(* CoDeSys 2.3.9.41 project: rePlc160.pro *)
(* Libraries: STANDARD.LIB 4.10.05 10:14:46, SmsOwenLib.lib 5.10.12 16:48:36, IECSFC.LIB 13.4.06 14:51:28, Util.lib 18.5.10 15:14:28, SysLibCom.lib 20.2.06 13:31:08, UNM.lib 14.2.06 12:27:08, SMS.lib 29.7.11 08:51:48, SYSLIBTIME.LIB 20.2.06 13:31:16, SYSTASKINFO.LIB 20.2.06 13:31:38, ANALYZATION.LIB 5.10.99 08:05:06, SYSLIBCALLBACK.LIB 20.2.06 13:31:08 *)

(* PLC configuration (modules and I/O channels)
DI_leakSens1 AT %IX0.0 [BitInput] Discrete input 1
DI_leakSens2 AT %IX0.1 [BitInput] Discrete input 2
DI_lamp1 AT %IX0.2 [BitInput] Discrete input 3
DI_lamp2 AT %IX0.3 [BitInput] Discrete input 4
AT %IB1.0 [ByteInput] DI_POLIW
AT %IB1.1 [ByteInput] DI_FOUNTAIN
AT %QB2.0 [ByteOutput] DO_POLIW_FOUN_LEAK
AT %QB2.1 [ByteOutput] DO_FOUN
AI_pres AT %IR3.0 [FloatInputP] AI #1 {AIN_TYPE = 0-20 mA; Peak_Filtr = 200; Flt_Ch = Off; TauRC = 10; MinFV = 0; MaxFV = 20000.0}
AI_level AT %IR3.1 [FloatInputP] AI #2 {AIN_TYPE = 0-20 mA; Peak_Filtr = 200; Flt_Ch = Off; TauRC = 10; MinFV = 0; MaxFV = 20000.0}
AI_T1 AT %IR3.2 [FloatInputP] AI #3 {AIN_TYPE = 4-20 mA; Peak_Filtr = 200; Flt_Ch = Off; TauRC = 10; MinFV = 0; MaxFV = 20000.0}
AI_T2 AT %IR3.3 [FloatInputP] AI #4 {AIN_TYPE = 4-20 mA; Peak_Filtr = 200; Flt_Ch = Off; TauRC = 10; MinFV = 0; MaxFV = 20000.0}
AI_05 AT %IR3.4 [FloatInputP] AI #5 {AIN_TYPE = 0-20 mA; Peak_Filtr = 200; Flt_Ch = Off; TauRC = 10; MinFV = 0; MaxFV = 20000.0}
AI_06 AT %IR3.5 [FloatInputP] AI #6 {AIN_TYPE = 0-20 mA; Peak_Filtr = 200; Flt_Ch = Off; TauRC = 10; MinFV = 0; MaxFV = 20000.0}
AI_volt AT %IR3.6 [FloatInputP] AI #7 {AIN_TYPE = 0-20 mA; Peak_Filtr = 200; Flt_Ch = Off; TauRC = 10; MinFV = 0; MaxFV = 20000.0}
AI_08 AT %IR3.7 [FloatInputP] AI #8 {AIN_TYPE = 0-20 mA; Peak_Filtr = 200; Flt_Ch = Off; TauRC = 10; MinFV = 0; MaxFV = 20000.0}
AT %IW3.8 [WordInput] AI read time (10ms)
AO_fc AT %QR4.0 [FloatOutputP] AO #1 {AOUT_TYPE = 0-10V; SafeValueREAL = 0.0}
AO_dim1 AT %QR4.1 [FloatOutputP] AO #2 {AOUT_TYPE = 0-10V; SafeValueREAL = 0.0}
AO_dim2 AT %QR4.2 [FloatOutputP] AO #3 {AOUT_TYPE = 0-10V; SafeValueREAL = 0.0}
AO_dim3 AT %QR4.3 [FloatOutputP] AO #4 {AOUT_TYPE = 0-10V; SafeValueREAL = 0.0}
Special input [ID103] node 5, in %IB5 out %QB5 {Filtrationtime = 1000; PinCount = 1; WatchDogPeriod = 400; PollPeriod = 3000; Visibility = No}
  AT %IX5.0 [BitInput] Special input
Special output [ID104] node 6, in %IB6 out %QB6 {Visibility = No; PinCount = 1}
  AT %QX6.0 [BitOutput] Special output
Universal network module [UNM_ID300] node 7, in %IB7 out %QB7 {Visibility = No}
  RS-232 [COM2_USART] node 0, in %IB7.0 out %QB7.0 {CommunicationSpeed = 9600; Parity = NO PARITY CHECK; BitLength = 8 bits; StopLength = One stop bit; InterfaceType = RS232; FrameOriented = ASCII; Timeout = 0; Visibility = No}
AT %QB8.0.0.0 [ByteOutput] Line Status
AT %QB8.0.0.1 [ByteOutput] Modem Fault
startGPRS AT %QB8.0.0.2 [ByteOutput] Start_Auto_Dial
stopGPRG AT %QB8.0.0.3 [ByteOutput] Stop_Dial
RS-232 [COM2_USART] node 0, in %IB8.0.0.0 out %QB8.0.0.0 {CommunicationSpeed = 9600; Parity = NO PARITY CHECK; BitLength = 8 bits; StopLength = One stop bit; InterfaceType = RS232; FrameOriented = ASCII; Timeout = 0; Visibility = No}
PPP_Driver [PPP] node 1, in %IB8.0.0.1 out %QB8.0.0.1 {LoginString = mts; PasswordString = mts}
TCP [TCP_ID221] node 1, in %IB8.0.1 out %QB8.0.1 {RemotePort = 502; Visibility = No}
pad_PoliwDIST AT %QW8.1.0 [WordOutput]
pad_PoliwTELE AT %QW8.2.0 [WordOutput]
cir1On AT %QW8.3.0 [WordOutput]
cir1Off AT %QW8.4.0 [WordOutput]
cir2On AT %QW8.5.0 [WordOutput]
2 byte [Register] node 6, in %IB8.6 out %QB8.6
  cir2Off AT %QW8.6.0 [WordOutput]
2 byte [Register] node 7, in %IB8.7 out %QB8.7
  cir3On AT %QW8.7.0 [WordOutput]
2 byte [Register] node 8, in %IB8.8 out %QB8.8
  cir3Off AT %QW8.8.0 [WordOutput]
  FounDIST AT %QW8.9.0 [WordOutput]
  dist_staticFValue AT %QW8.10.0 [WordOutput]
  FounTELE AT %QW8.11.0 [WordOutput]
  p1 AT %QW8.12.0 [WordOutput]
  p2 AT %QW8.13.0 [WordOutput]
2 byte [Register] node 14, in %IB8.14 out %QB8.14
  p3 AT %QW8.14.0 [WordOutput]
2 byte [Register] node 15, in %IB8.15 out %QB8.15
  p4 AT %QW8.15.0 [WordOutput]
2 byte [Register] node 16, in %IB8.16 out %QB8.16
  p5 AT %QW8.16.0 [WordOutput]
2 byte [Register] node 17, in %IB8.17 out %QB8.17
  p6 AT %QW8.17.0 [WordOutput]
2 byte [Register] node 18, in %IB8.18 out %QB8.18
  p7 AT %QW8.18.0 [WordOutput]
2 byte [Register] node 19, in %IB8.19 out %QB8.19
  p8 AT %QW8.19.0 [WordOutput]
2 byte [Register] node 20, in %IB8.20 out %QB8.20
  p9 AT %QW8.20.0 [WordOutput]
  p10 AT %QW8.21.0 [WordOutput]
2 byte [Register] node 22, in %IB8.22 out %QB8.22
  T_STATE AT %QW8.22.0 [WordOutput]
2 byte [Register] node 23, in %IB8.23 out %QB8.23
  pad_t1 AT %QW8.23.0 [WordOutput]
2 byte [Register] node 24, in %IB8.24 out %QB8.24
  pad_t2 AT %QW8.24.0 [WordOutput]
2 byte [Register] node 25, in %IB8.25 out %QB8.25
  pad_t1_currSetTop AT %QW8.25.0 [WordOutput]
2 byte [Register] node 26, in %IB8.26 out %QB8.26
  pad_t1_currSetBottom AT %QW8.26.0 [WordOutput]
2 byte [Register] node 27, in %IB8.27 out %QB8.27
  pad_t2_currSetTop AT %QW8.27.0 [WordOutput]
2 byte [Register] node 28, in %IB8.28 out %QB8.28
  pad_t2_currSetBottom AT %QW8.28.0 [WordOutput]
2 byte [Register] node 29, in %IB8.29 out %QB8.29
  pad_t1_day AT %QW8.29.0 [WordOutput]
2 byte [Register] node 30, in %IB8.30 out %QB8.30
  pad_t1_night AT %QW8.30.0 [WordOutput]
2 byte [Register] node 31, in %IB8.31 out %QB8.31
  pad_t2_day AT %QW8.31.0 [WordOutput]
2 byte [Register] node 32, in %IB8.32 out %QB8.32
  pad_t2_night AT %QW8.32.0 [WordOutput]
2 byte [Register] node 33, in %IB8.33 out %QB8.33
  pad_t1_daySetTop AT %QW8.33.0 [WordOutput]
2 byte [Register] node 34, in %IB8.34 out %QB8.34
  pad_t1_daySetBottom AT %QW8.34.0 [WordOutput]
2 byte [Register] node 35, in %IB8.35 out %QB8.35
  pad_t1_nightSetTop AT %QW8.35.0 [WordOutput]
2 byte [Register] node 36, in %IB8.36 out %QB8.36
  pad_t1_nightSetBottom AT %QW8.36.0 [WordOutput]
2 byte [Register] node 37, in %IB8.37 out %QB8.37
  pad_t2_daySetTop AT %QW8.37.0 [WordOutput]
2 byte [Register] node 38, in %IB8.38 out %QB8.38
  pad_t2_daySetBottom AT %QW8.38.0 [WordOutput]
  pad_t2_nightSetTop AT %QW8.39.0 [WordOutput]
  pad_t2_nightSetBottom AT %QW8.40.0 [WordOutput]
  pad_sens1_4ma AT %QW8.41.0 [WordOutput]
  pad_sens1_20ma AT %QW8.42.0 [WordOutput]
  pad_sens2_4ma AT %QW8.43.0 [WordOutput]
  pad_sens2_20ma AT %QW8.44.0 [WordOutput]
  dim1 AT %QW8.45.0 [WordOutput]
  dim2 AT %QW8.46.0 [WordOutput]
  dim3 AT %QW8.47.0 [WordOutput]
  RESERVE_1 AT %QW8.48.0 [WordOutput]
  RESERVE_2 AT %QW8.49.0 [WordOutput]
  weBITS_IN AT %QW8.50.0 [WordOutput] (leak)
  weBITS_OUT AT %QW8.51.0 [WordOutput] leakSens1,leakSens2,valveStat,drePumpStat,unknPump
  dist_LAMP AT %QW8.52.0 [WordOutput]
  tele_LAMP AT %QW8.53.0 [WordOutput]
  lamp1On AT %QW8.54.0 [WordOutput]
  lamp1Off AT %QW8.55.0 [WordOutput]
  lamp2On AT %QW8.56.0 [WordOutput]
  lamp2Off AT %QW8.57.0 [WordOutput]
  lamp3On AT %QW8.58.0 [WordOutput]
  lamp3Off AT %QW8.59.0 [WordOutput]
  year AT %QW8.60.0 [WordOutput]
  monthday AT %QW8.61.0 [WordOutput]
  hourminute AT %QW8.62.0 [WordOutput]
  tele_year AT %QW8.63.0 [WordOutput]
  tele_month AT %QW8.64.0 [WordOutput]
  tele_day AT %QW8.65.0 [WordOutput]
  tele_hour AT %QW8.66.0 [WordOutput]
  tele_minute AT %QW8.67.0 [WordOutput]
  dist_dom2 AT %QW8.68.0 [WordOutput]
  tele_dom2 AT %QW8.69.0 [WordOutput]
  tele_pres AT %QW8.70.0 [WordOutput]
  tele_level AT %QW8.71.0 [WordOutput]
  tele_voltage AT %QW8.72.0 [WordOutput]
*)

(* Global variable list: Global_Variables *)
VAR_GLOBAL

(* Times *)
	GetTime: CurTimeEx;
	TimeAndDate: SystemTimeDate;
	Sys_Time: SysTime64;

	SMS_ID  : WORD;

	DI_door : BOOL := FALSE;
	DO_door : BOOL := FALSE;
	DO_drePump : BOOL := FALSE;
	DO_unknownPump : BOOL := FALSE;
	DI_staticMode : BOOL := FALSE;
	DI_dynamicMode : BOOL := FALSE;
	DI_v1_manMode : BOOL := FALSE;
	DI_v2_manMode : BOOL := FALSE;
	DI_v3_manMode : BOOL := FALSE;
	DO_pump : BOOL := FALSE;
	DI_pumpState : BOOL := FALSE;

END_VAR

(* POU PLC_PRG, ST *)
PROGRAM PLC_PRG
VAR
	NO_FIRST_PASS : BOOL;
END_VAR
VAR RETAIN
	weBITS_IN_save : WORD;
END_VAR
IF NO_FIRST_PASS = FALSE
	THEN _WithdrawRetain;
	NO_FIRST_PASS := TRUE;
END_IF;

_CheckNewValue;

_Leakage;

_Tele;

POLIW;

FOUNTAIN;

TEMPERATURE;

LIGHT;

SMS;

DOM2;
END_PROGRAM
ACTION _CheckNewValue:
IF weBITS_IN_save <> weBITS_IN
	THEN weBITS_IN_save := weBITS_IN;
END_IF;
END_ACTION
ACTION _Leakage:
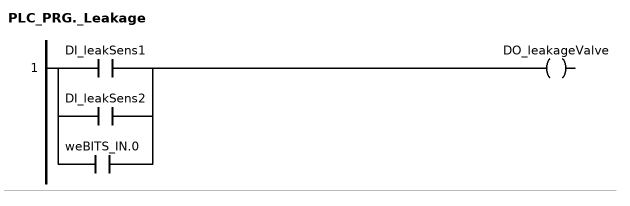
_LD_ (* Ladder Diagram *)
NETWORK 1
	{ [DI_leakSens1] | [DI_leakSens2] | [weBITS_IN.0] } --- (DO_leakageValve)
_END_LD_
(* the same logic as Structured Text *)
(* Network 1 *)
DO_leakageValve := DI_leakSens1 OR DI_leakSens2 OR weBITS_IN.0;
END_ACTION
ACTION _Tele:
weBITS_OUT.0 := DI_leakSens1;
weBITS_OUT.1 := DI_leakSens2;
weBITS_OUT.2 := DO_leakageValve;

(*
AI1_OUT := REAL_TO_WORD ( AI_01 );
AI2_OUT := REAL_TO_WORD ( AI_02 );
AI3_OUT := REAL_TO_WORD ( AI_T1 );
AI4_OUT := REAL_TO_WORD ( AI_T2 );
AI5_OUT := REAL_TO_WORD ( AI_05 );
AI6_OUT := REAL_TO_WORD ( AI_06 );
AI7_OUT := REAL_TO_WORD ( AI_07 );
AI8_OUT := REAL_TO_WORD ( AI_08 );
*)
(*
someDIs.0 := DI_konduk;
someDIs.1 := DI_powerSupply;
someDIs.2 := DI_banya;
someDIs.3 := DI_pool;
someDIs.4 := DI_foun;
someDIs.5 := DI_poliw;
someDIs.6 := DO_door;
*)
END_ACTION
ACTION _WithdrawRetain:
weBITS_IN := weBITS_IN_save;
END_ACTION

(* POU POLIW, ST *)
PROGRAM POLIW
VAR
	NO_FIRST_PASS : BOOL;
	PUNCH : WORD;
	setYear : INT;
	setMonth, setDay, setHour, setMinute : BYTE;
	set_time : BOOL;

(* bits *)
	dist_valve1, dist_valve2, dist_valve3 : BOOL;

	dist_manka : BOOL;

	MON : BOOL;
	TUE : BOOL;
	WED : BOOL;
	THU : BOOL;
	FRI : BOOL;
	SAT : BOOL;
	SUN : BOOL;

	cir1OnHH, cir1OnMM, cir1OffHH, cir1OffMM,
	cir2OnHH, cir2OnMM, cir2OffHH, cir2OffMM,
	cir3OnHH, cir3OnMM, cir3OffHH, cir3OffMM : BYTE;


	tele_pumpState, tele_v1state, tele_v2state, tele_v3state,
	tele_rainSens, tele_humSens : BOOL;

	cir1mustRun: BOOL;
	cir2mustRun: BOOL;
	cir3mustRun: BOOL;
	dayOk: BOOL;

	waterFault: BOOL;

	auto_pump_start: BOOL;
	auto_v1_open: BOOL;
	auto_v2_open: BOOL;
	auto_v3_open: BOOL;

	dist_pump_start: BOOL;
	dist_v1_open: BOOL;
	dist_v2_open: BOOL;
	dist_v3_open: BOOL;

	v1_auto_started: BOOL;
	FN_dist_v1_off: F_TRIG;
	v1_must_dist_stop: BOOL;
	v2_auto_started: BOOL;
	FN_dist_v2_off: F_TRIG;
	v2_must_dist_stop: BOOL;
	v3_auto_started: BOOL;
	FN_dist_v3_off: F_TRIG;
	v3_must_dist_stop: BOOL;
END_VAR

VAR RETAIN
	SAVE_BITS : WORD;

	save_cir1On, save_cir1Off,
       save_cir2On, save_cir2Off,
	 save_cir3On, save_cir3Off  : WORD;

	save_year, save_monthday, save_hourminute : WORD;
END_VAR
(* 				first pass 				*)
IF NO_FIRST_PASS = FALSE
	THEN WithdrawRetain;
	PUNCH := 65535;
	Obtaining;
	PUNCH := 0;
	NO_FIRST_PASS := TRUE;
END_IF;

(*			    main cycle		  		*)
PUNCH := 0;

set_time := weBITS_IN.1;
Times; (* получение текущего времени *)

CheckNewVal; (* проверка наличия новых значений переменных из модбас *)
				 (* и запись их в retain переменные *)
IF PUNCH > 0 THEN
	Obtaining; (* распаковка retain переменных в рабочие переменные *)
END_IF;

Schedule; (* основной цикл полива *)
(*
ExMech; (* управление исполнительным механизмом *)
*)
Outs; (* управление выходами контроллера на полив *)

HandOff;
Tele; (* передача рабочего состояния на верхний уровень *)
END_PROGRAM
ACTION CheckNewVal:
IF SAVE_BITS <> pad_PoliwDIST
	THEN SAVE_BITS := pad_PoliwDIST;
			PUNCH.0 := TRUE;
END_IF;



IF save_cir1On <> cir1On
	THEN save_cir1On := cir1On;
			PUNCH.1 := TRUE;
END_IF;

IF save_cir1Off <> cir1Off
	THEN save_cir1Off := cir1Off;
			PUNCH.2 := TRUE;
END_IF;


IF save_cir2On <> cir2On
	THEN save_cir2On := cir2On;
			PUNCH.3 := TRUE;
END_IF;

IF save_cir2Off <> cir2Off
	THEN save_cir2Off := cir2Off;
			PUNCH.4 := TRUE;
END_IF;


IF save_cir3On <> cir3On
	THEN save_cir3On := cir3On;
			PUNCH.5 := TRUE;
END_IF;

IF save_cir3Off <> cir3Off
	THEN save_cir3Off := cir3Off;
			PUNCH.6 := TRUE;
END_IF;


IF save_year <> year
	THEN save_year := year;
			PUNCH.9 := TRUE;
END_IF;

IF save_monthday <> monthday
	THEN save_monthday := monthday;
			PUNCH.10 := TRUE;
END_IF;

IF save_hourminute <> hourminute
	THEN save_hourminute := hourminute;
			PUNCH.11 := TRUE;
END_IF;
END_ACTION
ACTION HandOff:
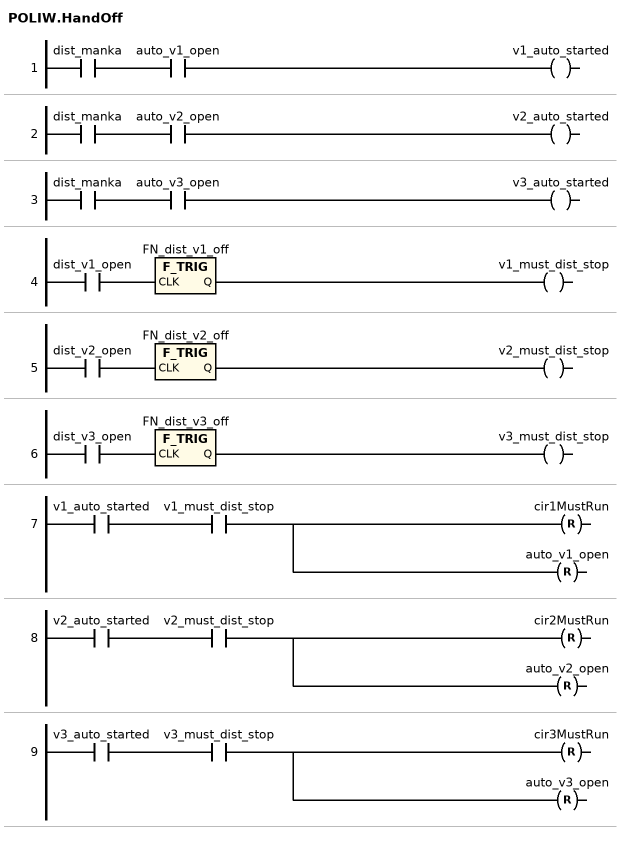
_LD_ (* Ladder Diagram *)
NETWORK 1
	[dist_manka] - [auto_v1_open] --- (v1_auto_started)
NETWORK 2
	[dist_manka] - [auto_v2_open] --- (v2_auto_started)
NETWORK 3
	[dist_manka] - [auto_v3_open] --- (v3_auto_started)
NETWORK 4
	[dist_v1_open] - FN_dist_v1_off:F_TRIG(CLK: *) --- (v1_must_dist_stop)
NETWORK 5
	[dist_v2_open] - FN_dist_v2_off:F_TRIG(CLK: *) --- (v2_must_dist_stop)
NETWORK 6
	[dist_v3_open] - FN_dist_v3_off:F_TRIG(CLK: *) --- (v3_must_dist_stop)
NETWORK 7
	[v1_auto_started] - [v1_must_dist_stop] --- (R cir1MustRun) (R auto_v1_open)
NETWORK 8
	[v2_auto_started] - [v2_must_dist_stop] --- (R cir2MustRun) (R auto_v2_open)
NETWORK 9
	[v3_auto_started] - [v3_must_dist_stop] --- (R cir3MustRun) (R auto_v3_open)
_END_LD_
(* the same logic as Structured Text *)
(* Network 1 *)
v1_auto_started := dist_manka AND auto_v1_open;
(* Network 2 *)
v2_auto_started := dist_manka AND auto_v2_open;
(* Network 3 *)
v3_auto_started := dist_manka AND auto_v3_open;
(* Network 4 *)
FN_dist_v1_off(CLK := dist_v1_open);
v1_must_dist_stop := FN_dist_v1_off.Q;
(* Network 5 *)
FN_dist_v2_off(CLK := dist_v2_open);
v2_must_dist_stop := FN_dist_v2_off.Q;
(* Network 6 *)
FN_dist_v3_off(CLK := dist_v3_open);
v3_must_dist_stop := FN_dist_v3_off.Q;
(* Network 7 *)
IF v1_auto_started AND v1_must_dist_stop THEN cir1MustRun := FALSE; auto_v1_open := FALSE; END_IF;
(* Network 8 *)
IF v2_auto_started AND v2_must_dist_stop THEN cir2MustRun := FALSE; auto_v2_open := FALSE; END_IF;
(* Network 9 *)
IF v3_auto_started AND v3_must_dist_stop THEN cir3MustRun := FALSE; auto_v3_open := FALSE; END_IF;
END_ACTION
ACTION Obtaining:
IF PUNCH.0 THEN
	dist_manka := SAVE_BITS.0;
	dist_valve1 := SAVE_BITS.1;
	dist_valve2 := SAVE_BITS.2;
	dist_valve3 := SAVE_BITS.3;

	MON := SAVE_BITS.6;
	TUE := SAVE_BITS.7;
	WED := SAVE_BITS.8;
	THU := SAVE_BITS.9;
	FRI := SAVE_BITS.10;
	SAT := SAVE_BITS.11;
	SUN := SAVE_BITS.12;

	PUNCH.0 := FALSE;
END_IF;

(*
	lo,hi : byte
	w : word

	lo := word_to_byte(w)
	hi := word_to_byte(w/256)
	w := 256*hi + lo 
*)

IF PUNCH.1 THEN
	cir1OnHH := WORD_TO_BYTE ( save_cir1On );
	cir1OnMM := WORD_TO_BYTE ( save_cir1On / 256 );
	PUNCH.1 := FALSE;
END_IF;

IF PUNCH.2 THEN
	cir1OffHH := WORD_TO_BYTE ( save_cir1Off );
	cir1OffMM := WORD_TO_BYTE ( save_cir1Off / 256 );
	PUNCH.2 := FALSE;
END_IF;

IF PUNCH.3 THEN
	cir2OnHH := WORD_TO_BYTE ( save_cir2On );
	cir2OnMM := WORD_TO_BYTE ( save_cir2On / 256 );
	PUNCH.3 := FALSE;
END_IF;

IF PUNCH.4 THEN
	cir2OffHH := WORD_TO_BYTE ( save_cir2Off );
	cir2OffMM := WORD_TO_BYTE ( save_cir2Off / 256 );
	PUNCH.4 := FALSE;
END_IF;

IF PUNCH.5 THEN
	cir3OnHH := WORD_TO_BYTE ( save_cir3On );
	cir3OnMM := WORD_TO_BYTE ( save_cir3On / 256 );
	PUNCH.5 := FALSE;
END_IF;

IF PUNCH.6 THEN
	cir3OffHH := WORD_TO_BYTE ( save_cir3Off );
	cir3OffMM := WORD_TO_BYTE ( save_cir3Off / 256 );
	PUNCH.6 := FALSE;
END_IF;


IF PUNCH.9 THEN
	setYear := WORD_TO_INT ( save_year );
	PUNCH.9 := FALSE;
END_IF;


IF PUNCH.10 THEN
	setDay := WORD_TO_BYTE ( save_monthday );
	setMonth := WORD_TO_BYTE ( save_monthday / 256 );
	PUNCH.10 := FALSE;
END_IF;

IF PUNCH.11 THEN
	setMinute := WORD_TO_BYTE ( save_hourminute );
	setHour := WORD_TO_BYTE ( save_hourminute / 256 );
	PUNCH.11 := FALSE;
END_IF;
END_ACTION
ACTION Outs:
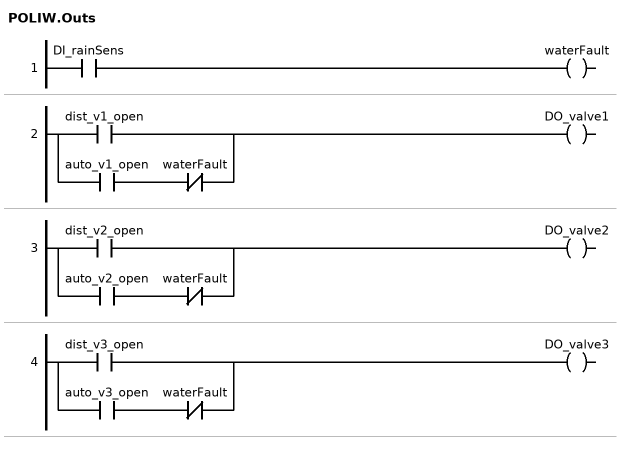
_LD_ (* Ladder Diagram *)
NETWORK 1
	[DI_rainSens] --- (waterFault)
NETWORK 2
	{ [dist_v1_open] | [auto_v1_open] - [/waterFault] } --- (DO_valve1)
NETWORK 3
	{ [dist_v2_open] | [auto_v2_open] - [/waterFault] } --- (DO_valve2)
NETWORK 4
	{ [dist_v3_open] | [auto_v3_open] - [/waterFault] } --- (DO_valve3)
_END_LD_
(* the same logic as Structured Text *)
(* Network 1 *)
waterFault := DI_rainSens;
(* Network 2 *)
DO_valve1 := dist_v1_open OR auto_v1_open AND NOT waterFault;
(* Network 3 *)
DO_valve2 := dist_v2_open OR auto_v2_open AND NOT waterFault;
(* Network 4 *)
DO_valve3 := dist_v3_open OR auto_v3_open AND NOT waterFault;
END_ACTION
ACTION Schedule:
(* контур 1 *)
IF ( cir1OnHH = TimeAndDate.Hour ) AND ( cir1OnMM = TimeAndDate.Minute ) AND ( TimeAndDate.Second = 0 )
	THEN cir1mustRun := TRUE;
END_IF;

IF ( cir1OffHH = TimeAndDate.Hour ) AND ( cir1OffMM = TimeAndDate.Minute ) AND ( TimeAndDate.Second = 0 )
	THEN cir1mustRun := FALSE;
END_IF;

(* контур 2 *)
IF ( cir2OnHH = TimeAndDate.Hour ) AND ( cir2OnMM = TimeAndDate.Minute ) AND ( TimeAndDate.Second = 0 )
	THEN cir2mustRun := TRUE;
END_IF;

IF ( cir2OffHH = TimeAndDate.Hour ) AND ( cir2OffMM = TimeAndDate.Minute ) AND ( TimeAndDate.Second = 0 )
	THEN cir2mustRun := FALSE;
END_IF;

(* контур 3 *)
IF ( cir3OnHH = TimeAndDate.Hour ) AND ( cir3OnMM = TimeAndDate.Minute ) AND ( TimeAndDate.Second = 0 )
	THEN cir3mustRun := TRUE;
END_IF;

IF ( cir3OffHH = TimeAndDate.Hour ) AND ( cir3OffMM = TimeAndDate.Minute ) AND ( TimeAndDate.Second = 0 )
	THEN cir3mustRun := FALSE;
END_IF;

(* день недели *)
CASE TimeAndDate.DayOfWeek OF
	1 : IF MON
	     	THEN dayOk := TRUE;
		ELSE dayOk := FALSE;
	     END_IF;

	2 : IF TUE
	     	THEN dayOk := TRUE;
		ELSE dayOk := FALSE;
	     END_IF;

      3 : IF WED
	     	THEN dayOk := TRUE;
		ELSE dayOk := FALSE;
	     END_IF;

      4 : IF THU
	     	THEN dayOk := TRUE;
		ELSE dayOk := FALSE;
	     END_IF;

      5 : IF FRI
	     	THEN dayOk := TRUE;
		ELSE dayOk := FALSE;
	     END_IF;

      6 : IF SAT
	     	THEN dayOk := TRUE;
		ELSE dayOk := FALSE;
	     END_IF;

      0 : IF SUN
	     	THEN dayOk := TRUE;
		ELSE dayOk := FALSE;
	     END_IF;
END_CASE;

(* авто *)
IF dist_manka = FALSE THEN
	(* клапана *)
	IF ( cir1mustRun ) AND ( dayOk )
		THEN auto_v1_open := TRUE;
		ELSE auto_v1_open := FALSE;
	END_IF;

	IF ( cir2mustRun ) AND ( dayOk )
		THEN auto_v2_open := TRUE;
		ELSE auto_v2_open := FALSE;
	END_IF;

	IF ( cir3mustRun ) AND ( dayOk )
		THEN auto_v3_open := TRUE;
		ELSE auto_v3_open := FALSE;
	END_IF;
END_IF;

(* ручное дистанционно *)
IF dist_manka  THEN
	IF dist_valve1
		THEN dist_v1_open := TRUE;
		ELSE dist_v1_open := FALSE;
	END_IF;

	IF dist_valve2
		THEN dist_v2_open := TRUE;
		ELSE dist_v2_open := FALSE;
	END_IF;

	IF dist_valve3
		THEN dist_v3_open := TRUE;
		ELSE dist_v3_open := FALSE;
	END_IF;
END_IF;

(* примечание: помимо дистанционного управления есть управление с галетников,
				   имеющее наивысший приоритет.
 				   управление с галетников описано в Outs 						

уже нет		*)
END_ACTION
ACTION Tele:
(*pad_PoliwTELE.0 := DI_pumpState;*)
pad_PoliwTELE.1 := DO_valve1;
pad_PoliwTELE.2 := DO_valve2;
pad_PoliwTELE.3 := DO_valve3;
(*pad_PoliwTELE.4 := DO_valve4;
pad_PoliwTELE.5 := DO_exMech;*)
pad_PoliwTELE.6 := DI_rainSens;
(*pad_PoliwTELE.7 := DI_humSens;*)

tele_year := TimeAndDate.Year;
tele_month := TimeAndDate.Month;
tele_day := TimeAndDate.Day;
tele_hour := TimeAndDate.Hour;
tele_minute := TimeAndDate.Minute;
END_ACTION
ACTION Times:
TimeAndDate.Day :=0;
TimeAndDate.DayOfWeek :=0;
TimeAndDate.dwHighMsec :=0;
TimeAndDate.dwLowMSecs :=0;
TimeAndDate.Milliseconds :=0;
TimeAndDate.Minute :=0;
TimeAndDate.Second :=0;
TimeAndDate.Hour :=0;
TimeAndDate.Year :=0;
TimeAndDate.Month :=0;
Sys_time.ulHigh :=0;
Sys_time.ulLow :=0;
GetTime (SystemTime:=Sys_Time , TimeDate:= TimeAndDate);


IF set_time THEN

	TimeAndDate.Minute:=setMinute;
	TimeAndDate.Second:=0;
	TimeAndDate.Hour:=setHour;
	TimeAndDate.Day:=setDay;
	TimeAndDate.Month:=setMonth;
	TimeAndDate.Year:=setYear;
	GetTime (SystemTime:=Sys_Time , TimeDate:= TimeAndDate);

END_IF;
END_ACTION
ACTION WithdrawRetain:
pad_PoliwDIST := SAVE_BITS;

cir1On := save_cir1On;
cir1Off := save_cir1Off;

cir2On := save_cir2On;
cir2Off := save_cir2Off;

cir3On := save_cir3On;
cir3Off := save_cir3Off;
END_ACTION

(* POU FOUNTAIN, ST *)
PROGRAM FOUNTAIN
VAR
	NO_FIRST_PASS : BOOL;
	PUNCH : WORD;

	tele_byte : BYTE;

	dist_founOn, dist_dynamic : BOOL;

	M1: BOOL;
	founT1: TON;
	M2: BOOL;
	founT2: TON;
	M3: BOOL;
	founT3: TON;
	M4: BOOL;
	founT4: TON;
	M5: BOOL;
	founT5: TON;
	M6: BOOL;
	founT6: TON;
	M7: BOOL;
	founT7: TON;
	M8: BOOL;
	founT8: TON;
	M9: BOOL;
	founT9: TON;
	M10: BOOL;
	founT10: TON;

	nodyn: BOOL;

	FPFON: R_TRIG;

	galetMode: BOOL;

(* ex-ratain*)
	staticFValue : REAL;

	founV1F: REAL;
	founV2F: REAL;
	founV3F: REAL;
	founV4F: REAL;
	founV5F: REAL;
	founV6F: REAL;
	founV7F: REAL;
	founV8F: REAL;
	founV9F: REAL;
	founV10F: REAL;

	founS1T: TIME;
	founS2T: TIME;
	founS3T: TIME;
	founS4T: TIME;
	founS5T: TIME;
	founS6T: TIME;
	founS7T: TIME;
	founS8T: TIME;
	founS9T: TIME;
	founS10T: TIME;
END_VAR

VAR RETAIN
	save_DIST : WORD;
	save_staticFValue : WORD;
	save_p1, save_p2, save_p3, save_p4, save_p5,
	save_p6, save_p7, save_p8, save_p9, save_p10 : WORD;

END_VAR
VAR (* helpers for the ST form of the networks *)
	_p1 : BOOL;
	_p2 : BOOL;
	_p3 : BOOL;
	_p4 : BOOL;
	_p5 : BOOL;
	_p6 : BOOL;
	_p7 : BOOL;
	_p8 : BOOL;
	_p9 : BOOL;
	_p10 : BOOL;
END_VAR
(* 				first pass 				*)
IF NO_FIRST_PASS = FALSE
	THEN WithdrawRetain;
	PUNCH := 1023;
	Obtaining;
	PUNCH := 0;
	NO_FIRST_PASS := TRUE;
END_IF;

(*			    main cycle		  		*)
PUNCH := 0;

CheckNewVal;

IF PUNCH > 0
	THEN Obtaining;
END_IF;


IF dist_dynamic
	THEN nodyn := FALSE;
	ELSE nodyn := TRUE;
END_IF;

IF ( founV1F = 0.0 ) AND
	( founV2F = 0.0 ) AND
	( founV3F = 0.0 ) AND
	( founV4F = 0.0 ) AND
	( founV5F = 0.0 ) AND
	( founV6F = 0.0 ) AND
	( founV7F = 0.0 ) AND
	( founV8F = 0.0 ) AND
	( founV9F = 0.0 ) AND
	( founV10F = 0.0 )
THEN
	nodyn := TRUE;
END_IF;

AOvalues;

PumpCtrl;

Forwarding;
END_PROGRAM
ACTION AOvalues:
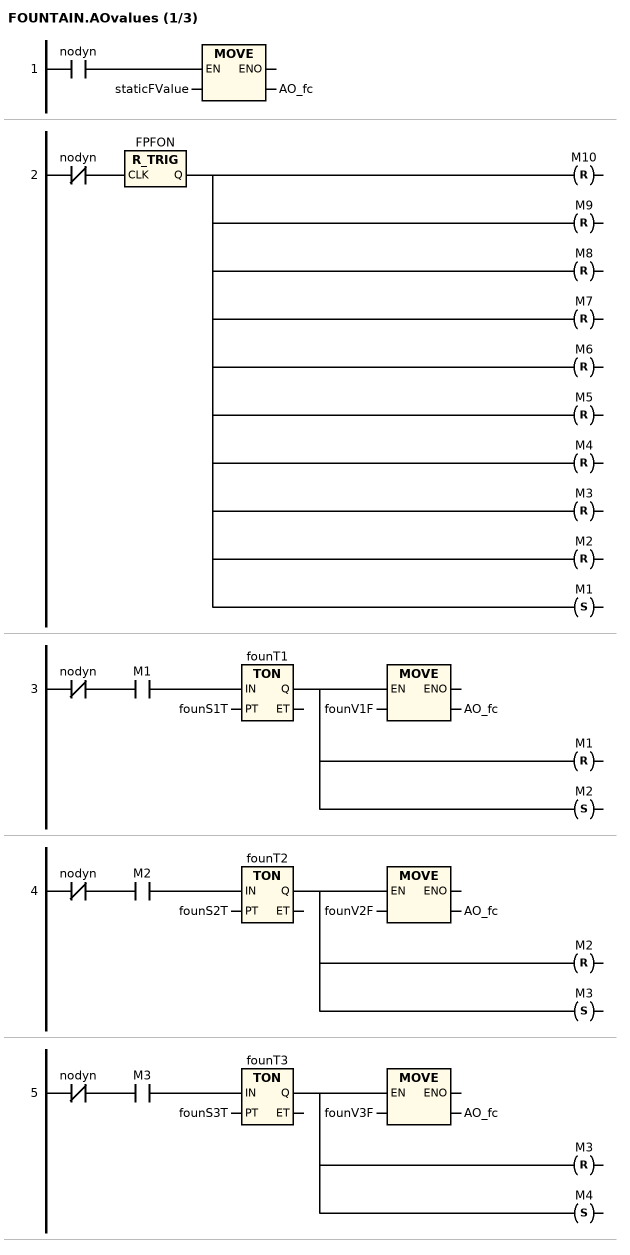
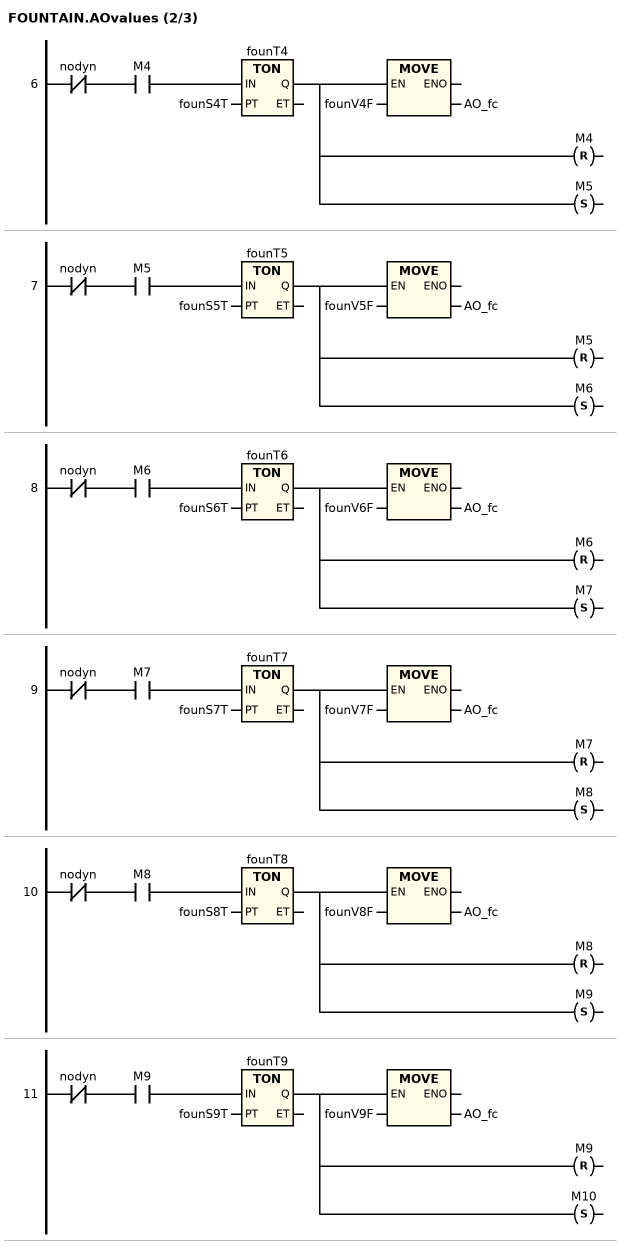
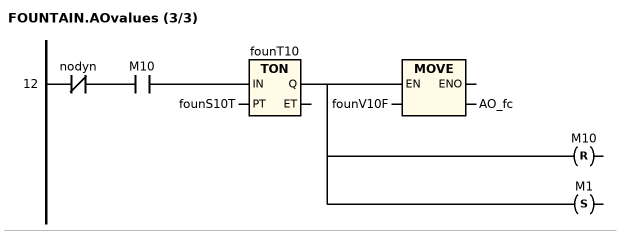
_LD_ (* Ladder Diagram *)
NETWORK 1
	[nodyn]
		EN --- MOVE(staticFValue) => AO_fc
NETWORK 2
	[/nodyn] - FPFON:R_TRIG(CLK: *) --- (R M10) (R M9) (R M8) (R M7) (R M6) (R M5) (R M4) (R M3) (R M2) (S M1)
NETWORK 3
	[/nodyn] - [M1] - founT1:TON(IN: *, PT: founS1T) --- (R M1) (S M2)
		EN --- MOVE(founV1F) => AO_fc
NETWORK 4
	[/nodyn] - [M2] - founT2:TON(IN: *, PT: founS2T) --- (R M2) (S M3)
		EN --- MOVE(founV2F) => AO_fc
NETWORK 5
	[/nodyn] - [M3] - founT3:TON(IN: *, PT: founS3T) --- (R M3) (S M4)
		EN --- MOVE(founV3F) => AO_fc
NETWORK 6
	[/nodyn] - [M4] - founT4:TON(IN: *, PT: founS4T) --- (R M4) (S M5)
		EN --- MOVE(founV4F) => AO_fc
NETWORK 7
	[/nodyn] - [M5] - founT5:TON(IN: *, PT: founS5T) --- (R M5) (S M6)
		EN --- MOVE(founV5F) => AO_fc
NETWORK 8
	[/nodyn] - [M6] - founT6:TON(IN: *, PT: founS6T) --- (R M6) (S M7)
		EN --- MOVE(founV6F) => AO_fc
NETWORK 9
	[/nodyn] - [M7] - founT7:TON(IN: *, PT: founS7T) --- (R M7) (S M8)
		EN --- MOVE(founV7F) => AO_fc
NETWORK 10
	[/nodyn] - [M8] - founT8:TON(IN: *, PT: founS8T) --- (R M8) (S M9)
		EN --- MOVE(founV8F) => AO_fc
NETWORK 11
	[/nodyn] - [M9] - founT9:TON(IN: *, PT: founS9T) --- (R M9) (S M10)
		EN --- MOVE(founV9F) => AO_fc
NETWORK 12
	[/nodyn] - [M10] - founT10:TON(IN: *, PT: founS10T) --- (R M10) (S M1)
		EN --- MOVE(founV10F) => AO_fc
_END_LD_
(* the same logic as Structured Text *)
(* Network 1 *)
IF nodyn THEN
	AO_fc := staticFValue;
END_IF;
(* Network 2 *)
FPFON(CLK := NOT nodyn);
IF FPFON.Q THEN M10 := FALSE; M9 := FALSE; M8 := FALSE; M7 := FALSE; M6 := FALSE; M5 := FALSE; M4 := FALSE; M3 := FALSE; M2 := FALSE; M1 := TRUE; END_IF;
(* Network 3 *)
founT1(IN := NOT nodyn AND M1, PT := founS1T);
_p1 := founT1.Q;
IF _p1 THEN
	AO_fc := founV1F;
END_IF;
IF _p1 THEN M1 := FALSE; M2 := TRUE; END_IF;
(* Network 4 *)
founT2(IN := NOT nodyn AND M2, PT := founS2T);
_p2 := founT2.Q;
IF _p2 THEN
	AO_fc := founV2F;
END_IF;
IF _p2 THEN M2 := FALSE; M3 := TRUE; END_IF;
(* Network 5 *)
founT3(IN := NOT nodyn AND M3, PT := founS3T);
_p3 := founT3.Q;
IF _p3 THEN
	AO_fc := founV3F;
END_IF;
IF _p3 THEN M3 := FALSE; M4 := TRUE; END_IF;
(* Network 6 *)
founT4(IN := NOT nodyn AND M4, PT := founS4T);
_p4 := founT4.Q;
IF _p4 THEN
	AO_fc := founV4F;
END_IF;
IF _p4 THEN M4 := FALSE; M5 := TRUE; END_IF;
(* Network 7 *)
founT5(IN := NOT nodyn AND M5, PT := founS5T);
_p5 := founT5.Q;
IF _p5 THEN
	AO_fc := founV5F;
END_IF;
IF _p5 THEN M5 := FALSE; M6 := TRUE; END_IF;
(* Network 8 *)
founT6(IN := NOT nodyn AND M6, PT := founS6T);
_p6 := founT6.Q;
IF _p6 THEN
	AO_fc := founV6F;
END_IF;
IF _p6 THEN M6 := FALSE; M7 := TRUE; END_IF;
(* Network 9 *)
founT7(IN := NOT nodyn AND M7, PT := founS7T);
_p7 := founT7.Q;
IF _p7 THEN
	AO_fc := founV7F;
END_IF;
IF _p7 THEN M7 := FALSE; M8 := TRUE; END_IF;
(* Network 10 *)
founT8(IN := NOT nodyn AND M8, PT := founS8T);
_p8 := founT8.Q;
IF _p8 THEN
	AO_fc := founV8F;
END_IF;
IF _p8 THEN M8 := FALSE; M9 := TRUE; END_IF;
(* Network 11 *)
founT9(IN := NOT nodyn AND M9, PT := founS9T);
_p9 := founT9.Q;
IF _p9 THEN
	AO_fc := founV9F;
END_IF;
IF _p9 THEN M9 := FALSE; M10 := TRUE; END_IF;
(* Network 12 *)
founT10(IN := NOT nodyn AND M10, PT := founS10T);
_p10 := founT10.Q;
IF _p10 THEN
	AO_fc := founV10F;
END_IF;
IF _p10 THEN M10 := FALSE; M1 := TRUE; END_IF;
END_ACTION
ACTION CheckNewVal:
IF save_DIST <> FounDIST
	THEN save_DIST:= FounDIST;
			PUNCH.0 := TRUE;
END_IF;

IF save_p1 <> p1
	THEN save_p1 := p1;
			PUNCH.1 := TRUE;
END_IF;

IF save_p2 <> p2
	THEN save_p2 := p2;
			PUNCH.2 := TRUE;
END_IF;

IF save_p3 <> p3
	THEN save_p3 := p3;
			PUNCH.3 := TRUE;
END_IF;

IF save_p4 <> p4
	THEN save_p4 := p4;
			PUNCH.4 := TRUE;
END_IF;

IF save_p5 <> p5
	THEN save_p5 := p5;
			PUNCH.5 := TRUE;
END_IF;

IF save_p6 <> p6
	THEN save_p6 := p6;
			PUNCH.6 := TRUE;
END_IF;

IF save_p7 <> p7
	THEN save_p7 := p7;
			PUNCH.7 := TRUE;
END_IF;

IF save_p8 <> p8
	THEN save_p8 := p8;
			PUNCH.8 := TRUE;
END_IF;

IF save_p9 <> p9
	THEN save_p9 := p9;
			PUNCH.9 := TRUE;
END_IF;

IF save_p10 <> p10
	THEN save_p10 := p10;
			PUNCH.10 := TRUE;
END_IF;

IF save_staticFValue <> dist_staticFValue
	THEN save_staticFValue := dist_staticFvalue;
			PUNCH.11 := TRUE;
END_IF;
END_ACTION
ACTION Forwarding:
(*
tele_byte.0 := DO_pump;
tele_byte.1 := DI_staticMode;
tele_byte.2 := DI_dynamicMode;
*)
FounTELE := REAL_TO_WORD ( AO_fc * 10 );
END_ACTION
ACTION Obtaining:
IF PUNCH.0 THEN
	dist_founOn := save_DIST.0;
	dist_dynamic := save_DIST.1;
(*
	staticFValue := BYTE_TO_REAL (
							WORD_TO_BYTE ( save_DIST / 256 ) ) / 10;
*)
	PUNCH.0 := FALSE;
END_IF;

IF PUNCH.11 THEN
	staticFValue := WORD_TO_REAL ( save_staticFValue ) / 10;
	PUNCH.11 := FALSE;
END_IF;

(*
	lo,hi : byte
	w : word

	lo := word_to_byte(w)
	hi := word_to_byte(w/256)
	w := 256*hi + lo 
*)

IF PUNCH.1 THEN
	founV1F := BYTE_TO_REAL ( WORD_TO_BYTE ( save_p1 ) ) / 10;
	founS1T := WORD_TO_TIME ( WORD_TO_BYTE ( save_p1 / 256 ) * 1000 );
	PUNCH.1 := FALSE;
END_IF;

IF PUNCH.2 THEN
	founV2F := BYTE_TO_REAL ( WORD_TO_BYTE ( save_p2 ) ) / 10;
	founS2T := WORD_TO_TIME ( WORD_TO_BYTE ( save_p2 / 256 ) * 1000 );
	PUNCH.2 := FALSE;
END_IF;

IF PUNCH.3 THEN
	founV3F := BYTE_TO_REAL ( WORD_TO_BYTE ( save_p3 ) ) /10;
	founS3T := WORD_TO_TIME ( WORD_TO_BYTE ( save_p3 / 256 ) * 1000 );
	PUNCH.3 := FALSE;
END_IF;

IF PUNCH.4 THEN
	founV4F := BYTE_TO_REAL ( WORD_TO_BYTE ( save_p4 ) ) /10;
	founS4T := WORD_TO_TIME ( WORD_TO_BYTE ( save_p4 / 256 ) * 1000 );
	PUNCH.4 := FALSE;
END_IF;

IF PUNCH.5 THEN
	founV5F := BYTE_TO_REAL ( WORD_TO_BYTE ( save_p5 ) ) /10;
	founS5T := WORD_TO_TIME ( WORD_TO_BYTE ( save_p5 / 256 ) * 1000 );
	PUNCH.5 := FALSE;
END_IF;

IF PUNCH.6 THEN
	founV6F := BYTE_TO_REAL ( WORD_TO_BYTE ( save_p6 ) ) /10;
	founS6T := WORD_TO_TIME ( WORD_TO_BYTE ( save_p6 / 256 ) * 1000 );
	PUNCH.6 := FALSE;
END_IF;

IF PUNCH.7 THEN
	founV7F := BYTE_TO_REAL ( WORD_TO_BYTE ( save_p7 ) ) /10;
	founS7T := WORD_TO_TIME ( WORD_TO_BYTE ( save_p7 / 256 ) * 1000 );
	PUNCH.7 := FALSE;
END_IF;

IF PUNCH.8 THEN
	founV8F := BYTE_TO_REAL ( WORD_TO_BYTE ( save_p8 ) ) /10;
	founS8T := WORD_TO_TIME ( WORD_TO_BYTE ( save_p8 / 256 ) * 1000 );
	PUNCH.8 := FALSE;
END_IF;

IF PUNCH.9 THEN
	founV9F := BYTE_TO_REAL ( WORD_TO_BYTE ( save_p9 ) ) /10;
	founS9T := WORD_TO_TIME ( WORD_TO_BYTE ( save_p9 / 256 ) * 1000 );
	PUNCH.9 := FALSE;
END_IF;

IF PUNCH.10 THEN
	founV10F := BYTE_TO_REAL ( WORD_TO_BYTE ( save_p10 ) ) /10;
	founS10T := WORD_TO_TIME ( WORD_TO_BYTE ( save_p10 / 256 ) * 1000 );
	PUNCH.10 := FALSE;
END_IF;
END_ACTION
ACTION PumpCtrl:
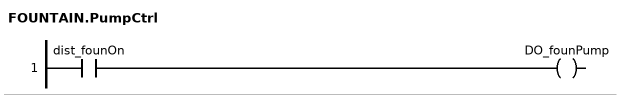
_LD_ (* Ladder Diagram *)
NETWORK 1
	[dist_founOn] --- (DO_founPump)
_END_LD_
(* the same logic as Structured Text *)
(* Network 1 *)
DO_founPump := dist_founOn;
END_ACTION
ACTION WithdrawRetain:
FounDIST := save_DIST;

p1 := save_p1;
p2 := save_p2;
p3 := save_p3;
p4 := save_p4;
p5 := save_p5;
p6 := save_p6;
p7 := save_p7;
p8 := save_p8;
p9 := save_p9;
p10 := save_p10;
END_ACTION

(* POU TEMPERATURE, ST *)
PROGRAM TEMPERATURE
VAR
	NO_FIRST_PASS : BOOL;
	tempOnCheck : TimeOnCheck;
	t1_out, t2_out : BOOL;
	t1_dayMode, t1_nightMode,
	t2_dayMode, t2_nightMode : BOOL;
	t1_topSet, t1_bottomSet,
	t2_topSet, t2_bottomSet : WORD;
	wordTemper1, wordTemper2 : WORD; (* точность 0.1 *)
END_VAR
VAR RETAIN
	t1_day, t1_night,
	t2_day, t2_night : WORD;

	t1_daySetTop, t1_daySetBottom,
       t1_nightSetTop, t1_nightSetBottom,
	t2_daySetTop, t2_daySetBottom,	(* точность 0.1 *)
       t2_nightSetTop, t2_nightSetBottom : WORD;

	sens1_4ma, sens1_20ma, (* точность 0.1 *)
	sens2_4ma, sens2_20ma : WORD;

END_VAR
(* 				first pass 				*)
IF NO_FIRST_PASS = FALSE
	THEN WithdrawRetain;
	Obtaining;
	NO_FIRST_PASS := TRUE;
END_IF;

Obtaining;

Schedule;

Calibration;

Setpoint;

Control;

Transfer;
END_PROGRAM
ACTION Calibration:
(*temperature := sens4ma / 100 + ( AI_02 / 1000 - 4 ) * ( ( sens20ma / 100 ) - ( sens4ma / 100 ) ) / 16;*)
(* точность до 0.1 *)
wordTemper1 := sens1_4ma + ( REAL_TO_WORD ( AI_T1 * 10 ) - 40 ) * ( sens1_20ma - sens1_4ma ) / 160;
wordTemper2 := sens2_4ma + ( REAL_TO_WORD ( AI_T2 * 10 ) - 40 ) * ( sens2_20ma - sens2_4ma ) / 160;
END_ACTION
ACTION Control:
IF wordTemper1 < t1_bottomSet THEN
	DO_heater1 := TRUE;
END_IF;

IF wordTemper1 > t1_topSet THEN
	DO_heater1 := FALSE;
END_IF;

IF wordTemper2 < t2_bottomSet THEN
	DO_heater2 := TRUE;
END_IF;

IF wordTemper2 > t2_topSet THEN
	DO_heater2 := FALSE;
END_IF;
END_ACTION
ACTION Obtaining:
t1_day    := pad_t1_day ;
t1_night := pad_t1_night;
t2_day    := pad_t2_day;
t2_night := pad_t2_night;

t1_daySetTop :=         pad_t1_daySetTop;
t1_daySetBottom :=   pad_t1_daySetBottom;
t1_nightSetTop :=       pad_t1_nightSetTop;
t1_nightSetBottom := pad_t1_nightSetBottom;

t2_daySetTop :=          pad_t2_daySetTop;
t2_daySetBottom :=    pad_t2_daySetBottom;
t2_nightSetTop :=       pad_t2_nightSetTop;
t2_nightSetBottom := pad_t2_nightSetBottom;
END_ACTION
ACTION Schedule:
tempOnCheck (
	currentState := t1_dayMode,
	needOffTime := TRUE,
	onTime := t1_day,
	offTime := t1_night,
	mustOn=> t1_dayMode
);

tempOnCheck (
		currentState := t1_nightMode,
		needOffTime := TRUE,
		onTime := t1_night,
		offTime := t1_day,
		mustOn=> t1_nightMode
);

tempOnCheck (
	currentState := t2_dayMode,
	needOffTime := TRUE,
	onTime := t2_day,
	offTime := t2_night,
	mustOn=> t2_dayMode
);

tempOnCheck (
		currentState := t2_nightMode,
		needOffTime := TRUE,
		onTime := t2_night,
		offTime := t2_day,
		mustOn=> t2_nightMode
);
END_ACTION
ACTION Setpoint:
IF t1_dayMode THEN
	t1_topSet := t1_daySetTop;
	t1_bottomSet := t1_daySetBottom;
END_IF;

IF t1_nightMode THEN
	t1_topSet := t1_nightSetTop;
	t1_bottomSet := t1_nightSetBottom;
END_IF;


IF t2_dayMode THEN
	t2_topSet := t2_daySetTop;
	t2_bottomSet := t2_daySetBottom;
END_IF;

IF t2_nightMode THEN
	t2_topSet := t2_nightSetTop;
	t2_bottomSet := t2_nightSetBottom;
END_IF;
END_ACTION
ACTION Transfer:
pad_t1 := wordTemper1;
pad_t2 := wordTemper2;

pad_t1_currSetTop := t1_topSet;
pad_t1_currSetBottom := t1_bottomSet;
pad_t2_currSetTop := t2_topSet;
pad_t2_currSetBottom := t2_bottomSet;

T_STATE.0 := DO_heater1;
T_STATE.1 := DO_heater2;
END_ACTION
ACTION WithdrawRetain:
pad_t1_day := t1_day;
pad_t1_night := t1_night;
pad_t2_day := t2_day;
pad_t2_night := t2_night;

pad_t1_daySetTop := t1_daySetTop;
pad_t1_daySetBottom := t1_daySetBottom;
pad_t1_nightSetTop := t1_nightSetTop;
pad_t1_nightSetBottom := t1_nightSetBottom;

pad_t2_daySetTop := t2_daySetTop;
pad_t2_daySetBottom := t2_daySetBottom;
pad_t2_nightSetTop := t2_nightSetTop;
pad_t2_nightSetBottom := t2_nightSetBottom;
END_ACTION

(* POU TimeOnCheck, ST *)
FUNCTION_BLOCK TimeOnCheck
VAR_INPUT
	currentState : BOOL;
	needOffTime : BOOL;
	onTime : WORD;
	offTime : WORD;
END_VAR
VAR_OUTPUT
	mustOn : BOOL;
END_VAR
VAR
	onHH, onMM : BYTE;
	offHH, offMM : BYTE;
END_VAR
mustOn := currentState;

onHH := WORD_TO_BYTE ( onTime );
onMM := WORD_TO_BYTE ( onTime / 256 );

offHH := WORD_TO_BYTE ( offTime );
offMM := WORD_TO_BYTE ( offTime / 256 );


IF ( onHH = TimeAndDate.Hour ) AND ( onMM = TimeAndDate.Minute ) AND ( TimeAndDate.Second = 0 )
	THEN mustOn := TRUE;
END_IF;

IF needOffTime THEN
	IF ( offHH = TimeAndDate.Hour ) AND ( offMM = TimeAndDate.Minute ) AND ( TimeAndDate.Second = 0 )
		THEN mustOn := FALSE;
	END_IF;
END_IF;
END_FUNCTION_BLOCK

(* POU LIGHT, ST *)
PROGRAM LIGHT
VAR
	NO_FIRST_PASS : BOOL;

	boolLamp1: BOOL;
	boolLamp2: BOOL;
	boolLamp3: BOOL;
	FP1: R_TRIG;
	FP2: R_TRIG;
	FP3: R_TRIG;
	FN1: F_TRIG;
	FP4: R_TRIG;
	FP5: R_TRIG;
	FP6: R_TRIG;
	FN2: F_TRIG;
	FP7: R_TRIG;
	FP8: R_TRIG;
	FP9: R_TRIG;
	FN3: F_TRIG;

	lamp1OnHH, lamp1OnMM, lamp1OffHH, lamp1OffMM,
	lamp2OnHH, lamp2OnMM, lamp2OffHH, lamp2OffMM,
	lamp3OnHH, lamp3OnMM, lamp3OffHH, lamp3OffMM : BYTE;
END_VAR
VAR RETAIN

	diBuf1: BOOL;
	mxBuf1: BOOL;
	mx1: BOOL;
	dx1: BOOL;

	diBuf2: BOOL;
	mxBuf2: BOOL;
	mx2: BOOL;
	dx2: BOOL;


	diBuf3: BOOL;
	mxBuf3: BOOL;
	mx3: BOOL;
	dx3: BOOL;

	preDoLamp1 : BOOL;
	timeDoLamp1: BOOL;

	preDoLamp2 : BOOL;
	timeDoLamp2: BOOL;

	preDoLamp3 : BOOL;
	timeDoLamp3: BOOL;


	dim1_save, dim2_save, dim3_save : WORD;

	lamp1On_save, lamp1Off_save, lamp2On_save, lamp2Off_save,
	lamp3On_save, lamp3Off_save : WORD;


END_VAR
VAR (* helpers for the ST form of the networks *)
	_p1 : BOOL;
	_p2 : BOOL;
	_p3 : BOOL;
	_p4 : BOOL;
	_p5 : BOOL;
	_p6 : BOOL;
	_p7 : BOOL;
	_p8 : BOOL;
	_p9 : BOOL;
	_p10 : BOOL;
	_p11 : BOOL;
	_p12 : BOOL;
END_VAR
IF NO_FIRST_PASS = FALSE
	THEN WithdrawRetain;
			NO_FIRST_PASS := TRUE;
END_IF;

CheckNewValue;

AO_dim1 := WORD_TO_REAL ( dim1 ) / 10;
AO_dim2 := WORD_TO_REAL ( dim2 ) / 10;
AO_dim3 := WORD_TO_REAL ( dim3 ) / 10;

UnpackTime;
Schedule;
Lamp1;
Lamp2;
Lamp3;

DistLamp;
ForwardLampState;
END_PROGRAM
ACTION CheckNewValue:
IF dim1_save <> dim1
	THEN dim1_save := dim1;
END_IF;

IF dim2_save <> dim2
	THEN dim2_save := dim2;
END_IF;

IF dim3_save <> dim3
	THEN dim3_save := dim3;
END_IF;

IF lamp1On_save <> lamp1On
	THEN lamp1On_save := lamp1On;
END_IF;


IF lamp1Off_save <> lamp1Off
	THEN lamp1Off_save := lamp1Off;
END_IF;

IF lamp2On_save <> lamp2On
	THEN lamp2On_save := lamp2On;
END_IF;


IF lamp2Off_save <> lamp2Off
	THEN lamp2Off_save := lamp2Off;
END_IF;

IF lamp3On_save <> lamp3On
	THEN lamp3On_save := lamp3On;
END_IF;


IF lamp3Off_save <> lamp3Off
	THEN lamp3Off_save := lamp3Off;
END_IF;
END_ACTION
ACTION DistLamp:
boolLamp1 := dist_LAMP.0;
boolLamp2 := dist_LAMP.1;
boolLamp3 := dist_LAMP.2;
END_ACTION
ACTION ForwardLampState:
tele_LAMP.0 := DO_lamp1;
tele_LAMP.1 := DO_lamp2;
tele_LAMP.2 := DO_lamp3;

tele_lamp.10 := DO_founPump;
END_ACTION
ACTION Lamp1:
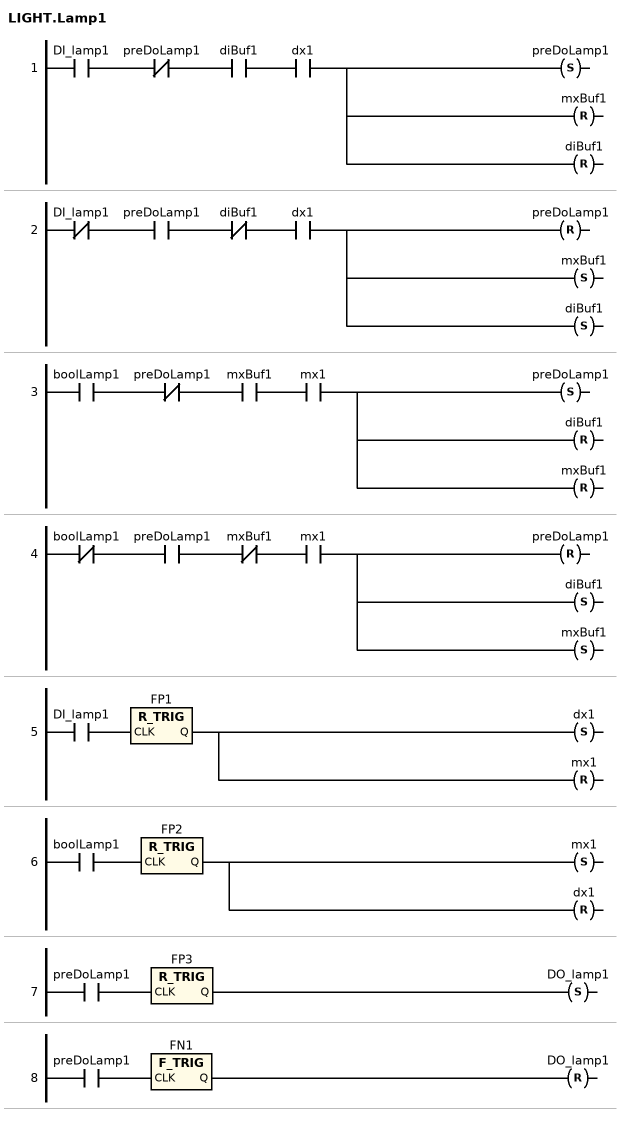
_LD_ (* Ladder Diagram *)
NETWORK 1
	[DI_lamp1] - [/preDoLamp1] - [diBuf1] - [dx1] --- (S preDoLamp1) (R mxBuf1) (R diBuf1)
NETWORK 2
	[/DI_lamp1] - [preDoLamp1] - [/diBuf1] - [dx1] --- (R preDoLamp1) (S mxBuf1) (S diBuf1)
NETWORK 3
	[boolLamp1] - [/preDoLamp1] - [mxBuf1] - [mx1] --- (S preDoLamp1) (R diBuf1) (R mxBuf1)
NETWORK 4
	[/boolLamp1] - [preDoLamp1] - [/mxBuf1] - [mx1] --- (R preDoLamp1) (S diBuf1) (S mxBuf1)
NETWORK 5
	[DI_lamp1] - FP1:R_TRIG(CLK: *) --- (S dx1) (R mx1)
NETWORK 6
	[boolLamp1] - FP2:R_TRIG(CLK: *) --- (S mx1) (R dx1)
NETWORK 7
	[preDoLamp1] - FP3:R_TRIG(CLK: *) --- (S DO_lamp1)
NETWORK 8
	[preDoLamp1] - FN1:F_TRIG(CLK: *) --- (R DO_lamp1)
_END_LD_
(* the same logic as Structured Text *)
(* Network 1 *)
_p1 := DI_lamp1 AND NOT preDoLamp1 AND diBuf1 AND dx1;
IF _p1 THEN preDoLamp1 := TRUE; mxBuf1 := FALSE; diBuf1 := FALSE; END_IF;
(* Network 2 *)
_p2 := NOT DI_lamp1 AND preDoLamp1 AND NOT diBuf1 AND dx1;
IF _p2 THEN preDoLamp1 := FALSE; mxBuf1 := TRUE; diBuf1 := TRUE; END_IF;
(* Network 3 *)
_p3 := boolLamp1 AND NOT preDoLamp1 AND mxBuf1 AND mx1;
IF _p3 THEN preDoLamp1 := TRUE; diBuf1 := FALSE; mxBuf1 := FALSE; END_IF;
(* Network 4 *)
_p4 := NOT boolLamp1 AND preDoLamp1 AND NOT mxBuf1 AND mx1;
IF _p4 THEN preDoLamp1 := FALSE; diBuf1 := TRUE; mxBuf1 := TRUE; END_IF;
(* Network 5 *)
FP1(CLK := DI_lamp1);
IF FP1.Q THEN dx1 := TRUE; mx1 := FALSE; END_IF;
(* Network 6 *)
FP2(CLK := boolLamp1);
IF FP2.Q THEN mx1 := TRUE; dx1 := FALSE; END_IF;
(* Network 7 *)
FP3(CLK := preDoLamp1);
IF FP3.Q THEN DO_lamp1 := TRUE; END_IF;
(* Network 8 *)
FN1(CLK := preDoLamp1);
IF FN1.Q THEN DO_lamp1 := FALSE; END_IF;
END_ACTION
ACTION Lamp2:
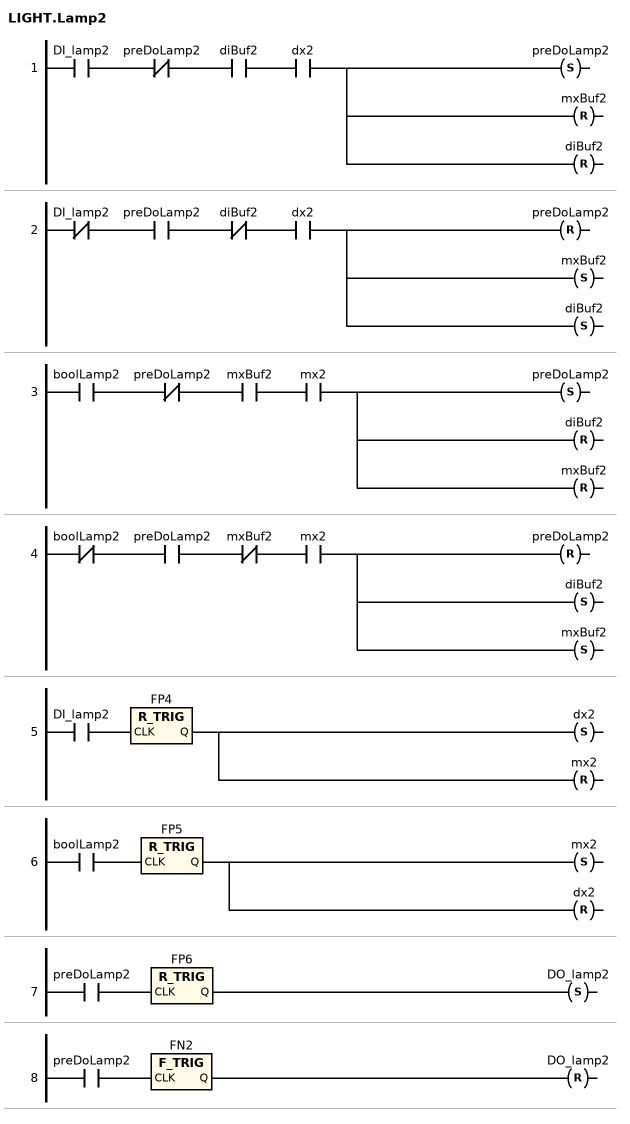
_LD_ (* Ladder Diagram *)
NETWORK 1
	[DI_lamp2] - [/preDoLamp2] - [diBuf2] - [dx2] --- (S preDoLamp2) (R mxBuf2) (R diBuf2)
NETWORK 2
	[/DI_lamp2] - [preDoLamp2] - [/diBuf2] - [dx2] --- (R preDoLamp2) (S mxBuf2) (S diBuf2)
NETWORK 3
	[boolLamp2] - [/preDoLamp2] - [mxBuf2] - [mx2] --- (S preDoLamp2) (R diBuf2) (R mxBuf2)
NETWORK 4
	[/boolLamp2] - [preDoLamp2] - [/mxBuf2] - [mx2] --- (R preDoLamp2) (S diBuf2) (S mxBuf2)
NETWORK 5
	[DI_lamp2] - FP4:R_TRIG(CLK: *) --- (S dx2) (R mx2)
NETWORK 6
	[boolLamp2] - FP5:R_TRIG(CLK: *) --- (S mx2) (R dx2)
NETWORK 7
	[preDoLamp2] - FP6:R_TRIG(CLK: *) --- (S DO_lamp2)
NETWORK 8
	[preDoLamp2] - FN2:F_TRIG(CLK: *) --- (R DO_lamp2)
_END_LD_
(* the same logic as Structured Text *)
(* Network 1 *)
_p5 := DI_lamp2 AND NOT preDoLamp2 AND diBuf2 AND dx2;
IF _p5 THEN preDoLamp2 := TRUE; mxBuf2 := FALSE; diBuf2 := FALSE; END_IF;
(* Network 2 *)
_p6 := NOT DI_lamp2 AND preDoLamp2 AND NOT diBuf2 AND dx2;
IF _p6 THEN preDoLamp2 := FALSE; mxBuf2 := TRUE; diBuf2 := TRUE; END_IF;
(* Network 3 *)
_p7 := boolLamp2 AND NOT preDoLamp2 AND mxBuf2 AND mx2;
IF _p7 THEN preDoLamp2 := TRUE; diBuf2 := FALSE; mxBuf2 := FALSE; END_IF;
(* Network 4 *)
_p8 := NOT boolLamp2 AND preDoLamp2 AND NOT mxBuf2 AND mx2;
IF _p8 THEN preDoLamp2 := FALSE; diBuf2 := TRUE; mxBuf2 := TRUE; END_IF;
(* Network 5 *)
FP4(CLK := DI_lamp2);
IF FP4.Q THEN dx2 := TRUE; mx2 := FALSE; END_IF;
(* Network 6 *)
FP5(CLK := boolLamp2);
IF FP5.Q THEN mx2 := TRUE; dx2 := FALSE; END_IF;
(* Network 7 *)
FP6(CLK := preDoLamp2);
IF FP6.Q THEN DO_lamp2 := TRUE; END_IF;
(* Network 8 *)
FN2(CLK := preDoLamp2);
IF FN2.Q THEN DO_lamp2 := FALSE; END_IF;
END_ACTION
ACTION Lamp3:
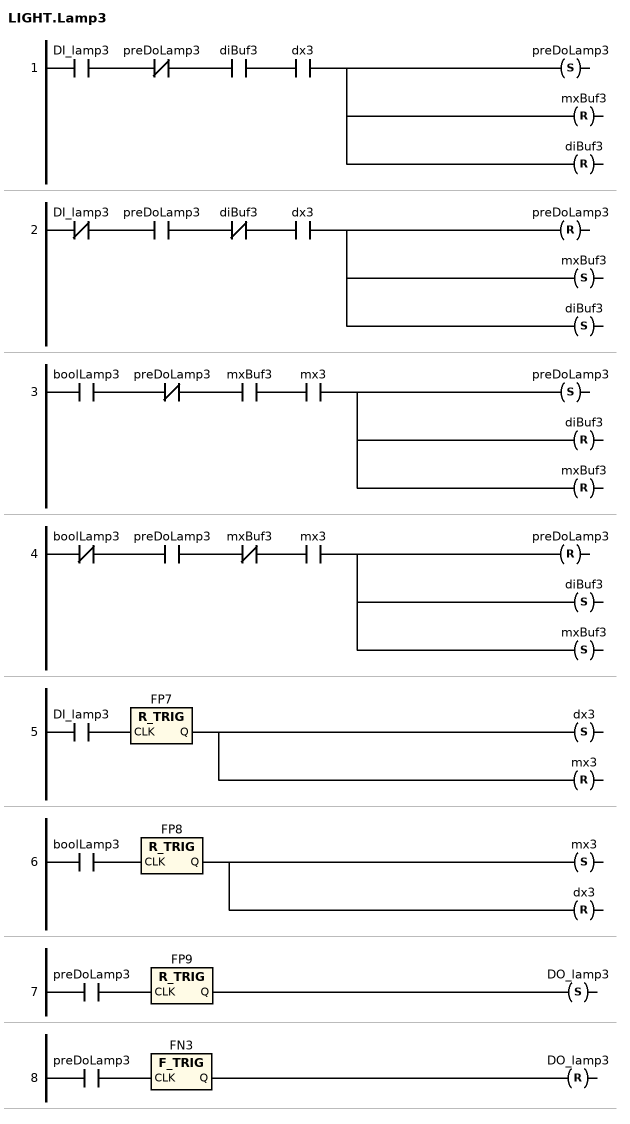
_LD_ (* Ladder Diagram *)
NETWORK 1
	[DI_lamp3] - [/preDoLamp3] - [diBuf3] - [dx3] --- (S preDoLamp3) (R mxBuf3) (R diBuf3)
NETWORK 2
	[/DI_lamp3] - [preDoLamp3] - [/diBuf3] - [dx3] --- (R preDoLamp3) (S mxBuf3) (S diBuf3)
NETWORK 3
	[boolLamp3] - [/preDoLamp3] - [mxBuf3] - [mx3] --- (S preDoLamp3) (R diBuf3) (R mxBuf3)
NETWORK 4
	[/boolLamp3] - [preDoLamp3] - [/mxBuf3] - [mx3] --- (R preDoLamp3) (S diBuf3) (S mxBuf3)
NETWORK 5
	[DI_lamp3] - FP7:R_TRIG(CLK: *) --- (S dx3) (R mx3)
NETWORK 6
	[boolLamp3] - FP8:R_TRIG(CLK: *) --- (S mx3) (R dx3)
NETWORK 7
	[preDoLamp3] - FP9:R_TRIG(CLK: *) --- (S DO_lamp3)
NETWORK 8
	[preDoLamp3] - FN3:F_TRIG(CLK: *) --- (R DO_lamp3)
_END_LD_
(* the same logic as Structured Text *)
(* Network 1 *)
_p9 := DI_lamp3 AND NOT preDoLamp3 AND diBuf3 AND dx3;
IF _p9 THEN preDoLamp3 := TRUE; mxBuf3 := FALSE; diBuf3 := FALSE; END_IF;
(* Network 2 *)
_p10 := NOT DI_lamp3 AND preDoLamp3 AND NOT diBuf3 AND dx3;
IF _p10 THEN preDoLamp3 := FALSE; mxBuf3 := TRUE; diBuf3 := TRUE; END_IF;
(* Network 3 *)
_p11 := boolLamp3 AND NOT preDoLamp3 AND mxBuf3 AND mx3;
IF _p11 THEN preDoLamp3 := TRUE; diBuf3 := FALSE; mxBuf3 := FALSE; END_IF;
(* Network 4 *)
_p12 := NOT boolLamp3 AND preDoLamp3 AND NOT mxBuf3 AND mx3;
IF _p12 THEN preDoLamp3 := FALSE; diBuf3 := TRUE; mxBuf3 := TRUE; END_IF;
(* Network 5 *)
FP7(CLK := DI_lamp3);
IF FP7.Q THEN dx3 := TRUE; mx3 := FALSE; END_IF;
(* Network 6 *)
FP8(CLK := boolLamp3);
IF FP8.Q THEN mx3 := TRUE; dx3 := FALSE; END_IF;
(* Network 7 *)
FP9(CLK := preDoLamp3);
IF FP9.Q THEN DO_lamp3 := TRUE; END_IF;
(* Network 8 *)
FN3(CLK := preDoLamp3);
IF FN3.Q THEN DO_lamp3 := FALSE; END_IF;
END_ACTION
ACTION Schedule:
(* 1 *)
IF ( lamp1OnHH = TimeAndDate.Hour ) AND ( lamp1OnMM = TimeAndDate.Minute ) AND ( TimeAndDate.Second = 0 )
	THEN DO_lamp1 := TRUE;
END_IF;

IF ( lamp1OffHH = TimeAndDate.Hour ) AND ( lamp1OffMM = TimeAndDate.Minute ) AND ( TimeAndDate.Second = 0 )
	THEN DO_lamp1 := FALSE;
END_IF;

(* 2 *)
IF ( lamp2OnHH = TimeAndDate.Hour ) AND ( lamp2OnMM = TimeAndDate.Minute ) AND ( TimeAndDate.Second = 0 )
	THEN DO_lamp2 := TRUE;
END_IF;

IF ( lamp2OffHH = TimeAndDate.Hour ) AND ( lamp2OffMM = TimeAndDate.Minute ) AND ( TimeAndDate.Second = 0 )
	THEN DO_lamp2 := FALSE;
END_IF;

(* 3 *)
IF ( lamp3OnHH = TimeAndDate.Hour ) AND ( lamp3OnMM = TimeAndDate.Minute ) AND ( TimeAndDate.Second = 0 )
	THEN DO_lamp3 := TRUE;
END_IF;

IF ( lamp3OffHH = TimeAndDate.Hour ) AND ( lamp3OffMM = TimeAndDate.Minute ) AND ( TimeAndDate.Second = 0 )
	THEN DO_lamp3 := FALSE;
END_IF;
END_ACTION
ACTION UnpackTime:
(*
	lo,hi : byte
	w : word

	lo := word_to_byte(w)
	hi := word_to_byte(w/256)
	w := 256*hi + lo 
*)
	lamp1OnHH := WORD_TO_BYTE ( lamp1On );
	lamp1OnMM := WORD_TO_BYTE ( lamp1On / 256 );

	lamp1OffHH := WORD_TO_BYTE ( lamp1Off );
	lamp1OffMM := WORD_TO_BYTE ( lamp1Off / 256 );


	lamp2OnHH := WORD_TO_BYTE ( lamp2On );
	lamp2OnMM := WORD_TO_BYTE ( lamp2On / 256 );

	lamp2OffHH := WORD_TO_BYTE ( lamp2Off );
	lamp2OffMM := WORD_TO_BYTE ( lamp2Off / 256 );


	lamp3OnHH := WORD_TO_BYTE ( lamp3On );
	lamp3OnMM := WORD_TO_BYTE ( lamp3On / 256 );

	lamp3OffHH := WORD_TO_BYTE ( lamp3Off );
	lamp3OffMM := WORD_TO_BYTE ( lamp3Off / 256 );
END_ACTION
ACTION WithdrawRetain:
dim1 := dim1_save;
dim2 := dim2_save;
dim3 := dim3_save;

lamp1On := lamp1On_save;
lamp1Off := lamp1Off_save;
lamp2On := lamp2On_save;
lamp2Off := lamp2Off_save;
lamp3On := lamp3On_save;
lamp3Off := lamp3Off_save;
END_ACTION

(* POU SMS, ST *)
PROGRAM SMS
VAR
	Com		: OpenPort;
	cfg		       : FB_SMS_CFG;
	sms		:FB_SMS_SR;
	cfg_ok		: BOOL := FALSE;
	sendSMS  : BOOL := FALSE;
	ready		: BOOL;
	DevNum	: WORD := 0;
	openModemPort : BOOL := FALSE;
	port_ok      : BOOL := FALSE;
	errCode     : BYTE;
	errBool      : BOOL;

	sendText   : STRING(70);
	sended     : BOOL;

	senderErrCode : BYTE;
	timeOut : TON;

	lock1, lock2, lock3, lock4 : BOOL := FALSE;
END_VAR
Inputs;

IF SMS_ID > 0 THEN
	Select;
	openModemPort := TRUE;
	sendSMS := TRUE;
ELSE
	openModemPort := FALSE;
	sendSMS := FALSE;
END_IF;

Configure;

IF ( cfg_ok=TRUE ) AND ( errBool=FALSE ) THEN

	ready := TRUE;
ELSE
	ready := FALSE;
END_IF;

Send;

IF sended THEN
	SMS_ID := 0;
	sendSMS := FALSE;
END_IF;

Timeout;
END_PROGRAM
ACTION Configure:
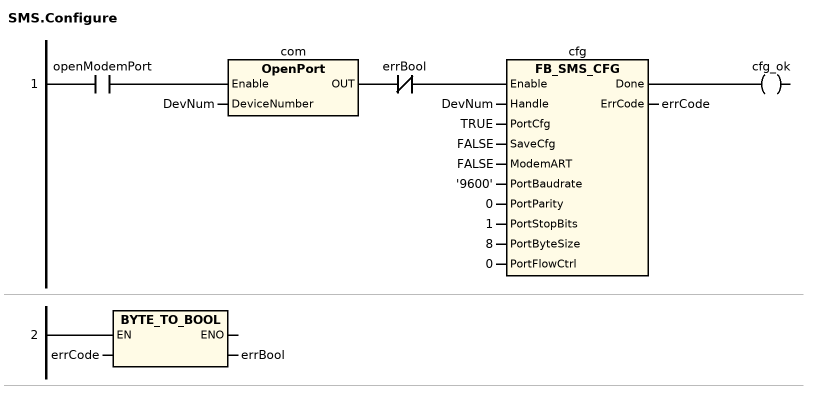
_LD_ (* Ladder Diagram *)
NETWORK 1
	[openModemPort] - com:OpenPort(Enable: *, DeviceNumber: DevNum) - [/errBool] - cfg:FB_SMS_CFG(Enable: *, Handle: DevNum, PortCfg: TRUE, SaveCfg: FALSE, ModemART: FALSE, PortBaudrate: '9600', PortParity: 0, PortStopBits: 1, PortByteSize: 8, PortFlowCtrl: 0, ErrCode => errCode) --- (cfg_ok)
NETWORK 2
	*
		EN --- BYTE_TO_BOOL(errCode) => errBool
_END_LD_
(* the same logic as Structured Text *)
(* Network 1 *)
com(Enable := openModemPort, DeviceNumber := DevNum);
cfg(Enable := com.OUT AND NOT errBool, Handle := DevNum, PortCfg := TRUE, SaveCfg := FALSE, ModemART := FALSE, PortBaudrate := '9600', PortParity := 0, PortStopBits := 1, PortByteSize := 8, PortFlowCtrl := 0);
errCode := cfg.ErrCode;
cfg_ok := cfg.Done;
(* Network 2 *)
errBool := BYTE_TO_BOOL(errCode);
END_ACTION
ACTION Inputs:
IF SMS_ID = 0 THEN
	IF DI_powerSupply AND lock1=FALSE THEN
		SMS_ID := 1;
		lock1 := TRUE;
	END_IF;
	IF DI_signal1 AND lock2=FALSE THEN
		SMS_ID := 2;
		lock2 := TRUE;
	END_IF;
	IF DI_signal2 AND lock3=FALSE THEN
		SMS_ID := 4;
		lock3 := TRUE;
	END_IF;
	IF DI_fireSignal AND lock4=FALSE THEN
		SMS_ID := 8;
		lock4 := TRUE;
	END_IF;
END_IF;

IF DI_powerSupply=FALSE THEN
	lock1 := FALSE;
END_IF;
IF DI_signal1=FALSE THEN
	lock2 := FALSE;
END_IF;
IF DI_signal2=FALSE THEN
	lock3 := FALSE;
END_IF;
IF DI_fireSignal=FALSE THEN
	lock4 := FALSE;
END_IF;
END_ACTION
ACTION Select:
IF SMS_ID.0 THEN
	sendText := 'Блок питания';
END_IF;

IF SMS_ID.1 THEN
	sendText := 'Извещатель охранный';
END_IF;

IF SMS_ID.2 THEN
	sendText := 'Извещатель объёмный';
END_IF;

IF SMS_ID.3 THEN
	sendText := 'Извещатель пожарный дымовой';
END_IF;
END_ACTION
ACTION Send:
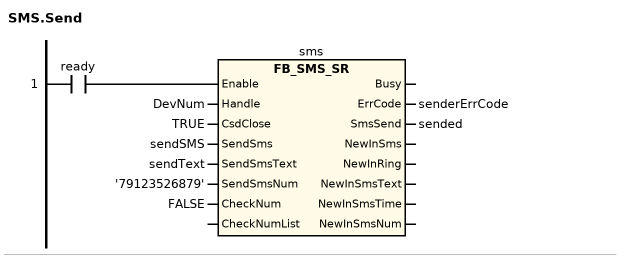
_LD_ (* Ladder Diagram *)
NETWORK 1
	[ready] - sms:FB_SMS_SR(Enable: *, Handle: DevNum, CsdClose: TRUE, SendSms: sendSMS, SendSmsText: sendText, SendSmsNum: '79123526879', CheckNum: FALSE, CheckNumList: , ErrCode => senderErrCode, SmsSend => sended)
_END_LD_
END_ACTION
ACTION Timeout:
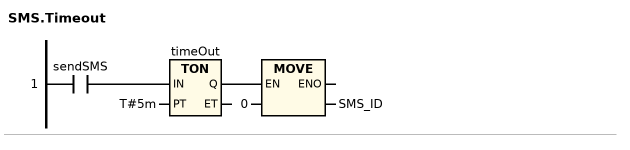
_LD_ (* Ladder Diagram *)
NETWORK 1
	[sendSMS] - timeOut:TON(IN: *, PT: T#5m)
		EN --- MOVE(0) => SMS_ID
_END_LD_
(* the same logic as Structured Text *)
(* Network 1 *)
timeOut(IN := sendSMS, PT := T#5m);
IF timeOut.Q THEN
	SMS_ID := 0;
END_IF;
END_ACTION

(* POU DOM2, ST *)
PROGRAM DOM2
VAR
END_VAR
DO_voltSupply := dist_dom2.0;
DO_banya := dist_dom2.1;

tele_dom2.0 := DI_powerSupply;
tele_dom2.1 := DO_banya;

tele_dom2.2 := DI_signal1;
tele_dom2.3 := DI_signal2;
tele_dom2.4 := DI_fireSignal;

tele_pres := REAL_TO_WORD( AI_pres * 1000 );
tele_level := REAL_TO_WORD( AI_level  );
tele_voltage := REAL_TO_WORD( AI_volt * 10 );
END_PROGRAM
